(* Logix 5000 project; controller Lab_PAC_Sensores vendor 1 type 14 code 156 rev 30.11; software revision 30.00 *)
// Práctica usando los PAC del laboratorio de automatización UNAL 2023/1

TASK MainTask (continuous, watchdog 500 ms) : MainProgram

MODULES
   Local : vendor 1 type 14 code 156 (Compact 0, rev 30.11)
      Ent_digital : 1769-IQ16 (Compact 4, rev 1.1, Input RPI 20 ms)   // Módulo de entradas digitales
      Sal_digital : vendor 1 type 7 code 86 (Compact 5, rev 2.1, Output RPI 20 ms)   // Módulo de salidas digitales
END_MODULES

PROGRAM MainProgram   (* main routine MainRoutine *)
VAR
   A_ev : BOOL;   // Forzar A+
   A_ext : ALIAS FOR Local:5:O.Data.0;   // Extender cilindro A
   A_ret : ALIAS FOR Local:5:O.Data.2;   // Retraer cilindro A
   A_rv : BOOL;   // Forzar A-
   B_ext : ALIAS FOR Local:5:O.Data.4;   // Extender cilindro B
   Counter1 : COUNTER := (PRE := 1, ACC := 1, DN := 1);   // Contador del cilindro B (conflicto)
   Counter2 : COUNTER := (PRE := 1);   // Bug
   Gaby : ALIAS FOR Local:4:I.Data.6;
   S1 : ALIAS FOR Local:4:I.Data.2;   // Sensor cilindro A ret
   S2 : ALIAS FOR Local:4:I.Data.3;   // Sensor cilindro A ext
   S3 : ALIAS FOR Local:4:I.Data.4;   // Sensor cilindro B ret
   S4 : ALIAS FOR Local:4:I.Data.5;   // Sensor cilindro B ext
   Start : ALIAS FOR Local:4:I.Data.1;   // Botón de arranque de secuencia
   Stop : ALIAS FOR Local:4:I.Data.0;   // Botón de parada de secuencia
   Tmr1 : TIMER := (PRE := 5000);
END_VAR

ROUTINE MainRoutine   (* ladder *)
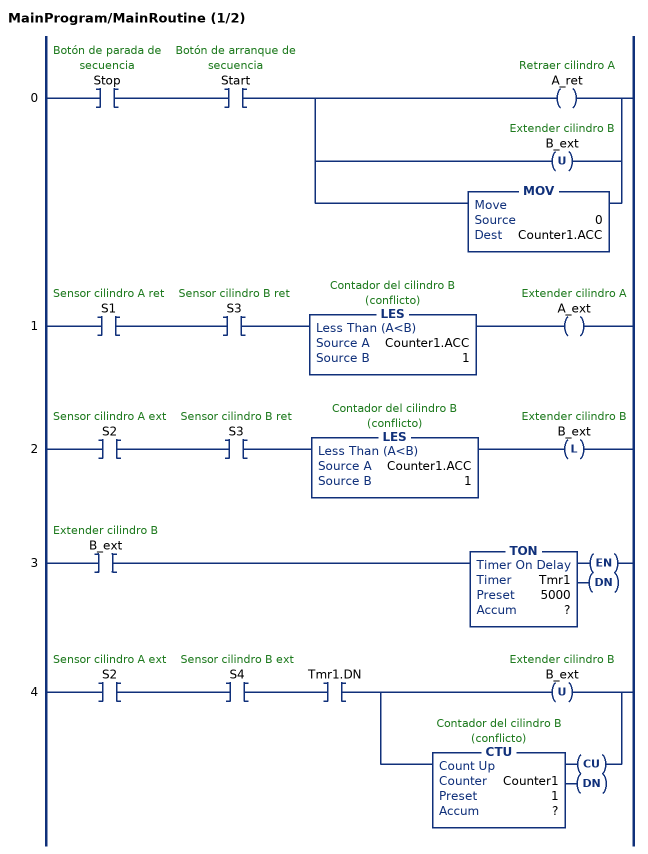
   0: XIC(Stop)XIC(Start)[OTE(A_ret) ,OTU(B_ext) ,MOV(0,Counter1.ACC) ];
   1: XIC(S1)XIC(S3)LES(Counter1.ACC,1)OTE(A_ext);
   2: XIC(S2)XIC(S3)LES(Counter1.ACC,1)OTL(B_ext);
   3: XIC(B_ext)TON(Tmr1,?,?);
   4: XIC(S2)XIC(S4)XIC(Tmr1.DN)[OTU(B_ext) ,CTU(Counter1,?,?) ];
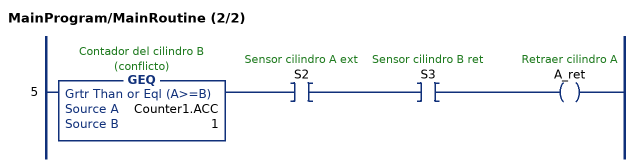
   5: GEQ(Counter1.ACC,1)XIC(S2)XIC(S3)OTE(A_ret);
END_ROUTINE
END_PROGRAM
